{attribute 'qualified_only'}
VAR_GLOBAL
	//OPC Bridge Heartbeat -- Logic found in heartbeat routine
	{attribute 'OPC.UA.DA' :='1'}
	opc_bridge_heartbeat : INT;
END_VAR

(* stored: Version 1.1.0.1, ProductVersion 3.1.4024.15
   GVL heartbeat: Id {c177fba1-82db-4009-ade4-95c277f10d8f} *)
